FUNCTION_BLOCK FB_MovingHead
VAR
	_Active : BOOL;
END_VAR

PROPERTY Active : BOOL
GET
Active := This^._Active;
END_GET
END_PROPERTY

METHOD Off : BOOL
VAR_INPUT
END_VAR
This^._Active := FALSE;
END_METHOD

METHOD On : BOOL
VAR_INPUT
END_VAR
This^._Active := TRUE;
END_METHOD

END_FUNCTION_BLOCK

(* stored: Version 1.1.0.1, ProductVersion 3.1.4022.18
   POU FB_MovingHead: Id {1cf169f5-f4e6-4495-923b-c7833b6dbc27}, SpecialFunc None
   Property Active: Id {47abe765-e271-4d93-87b2-8a42364c47b2}
   Get Get: Id {9bd35d94-b569-443d-80c1-ca3343c5b640}
   Method Off: Id {dd99ceb8-315b-45bb-91ee-ae819441b968}
   Method On: Id {e65ae756-3296-47fb-a145-de6c1d7346ec} *)
